FUNCTION_BLOCK FB_Axis
VAR_INPUT
END_VAR
VAR_OUTPUT
END_VAR
VAR
	bJogFwd			: BOOL;
	bJogRev			: BOOL;
	bFaulted		: BOOL;
	fPosition		: LREAL;
	fVelocity		: LREAL;
END_VAR

IF bJogFwd THEN
	fVelocity := 10.0;
	fPosition := fPosition + 0.1;
ELSE
	fVelocity := 0;
END_IF

IF bJogRev THEN
	fVelocity := -10.0;
	fPosition := fPosition - 0.1;
ELSE
	fVelocity := 0;
END_IF

END_FUNCTION_BLOCK

(* stored: Version 1.1.0.1, ProductVersion 3.1.4024.12
   POU FB_Axis: Id {de781bb2-1a71-409c-b7e0-37acf511f379}, SpecialFunc None *)
